// TIA Portal V20 export
FUNCTION_BLOCK "FB_FeedOverride"   // FB82, SCL
{ S7_Optimized_Access := 'TRUE' }
// stored: MemoryReserve 100, SetENOAutomatically false
   VAR_INPUT
      iA_FD_OR : Byte;
   END_VAR
   VAR_OUTPUT
      oFeedOverride : Byte;
   END_VAR
BEGIN
   REGION Description header 
       //==================================================================================
       // POSALUX Swiss SA / (C) Copyright 2026
       //----------------------------------------------------------------------------------
       // Title: FB_FeedObverride
       // Comment/Function: 
       // Author: Fabien WALDT
       // Engineering: TIA Portal v20
       //----------------------------------------------------------------------------------
       // Change log table:
       // Version  | Date     | Expert in charge | Changes applied
       // ---------|----------|------------------|-----------------------------------------
       // 00.00.01 | 20260309 | WFA              | First released version
       // =================================================================================
   END_REGION

   REGION Feed Ovr Value
       CASE #iA_FD_OR OF
           1:
               #oFeedOverride := 0;
           3:
               #oFeedOverride := 1;
           2:
               #oFeedOverride := 2;
           6:
               #oFeedOverride := 4;
           7:
               #oFeedOverride := 6;
           5:
               #oFeedOverride := 8;
           4:
               #oFeedOverride := 10;
           12:
               #oFeedOverride := 20;
           13:
               #oFeedOverride := 30;
           15:
               #oFeedOverride := 40;
           14:
               #oFeedOverride := 50;
           10:
               #oFeedOverride := 60;
           11:
               #oFeedOverride := 70;
           9:
               #oFeedOverride := 75;
           8:
               #oFeedOverride := 80;
           24:
               #oFeedOverride := 85;
           25:
               #oFeedOverride := 90;
           27:
               #oFeedOverride := 95;
           26:
               #oFeedOverride := 100;
           30:
               #oFeedOverride := 105;
           31:
               #oFeedOverride := 110;
           29:
               #oFeedOverride := 115;
           28:
               #oFeedOverride := 120;
       END_CASE;
   END_REGION
END_FUNCTION_BLOCK
